(* IEC 61131-3 sources: teller/JD_Teller_LC2_V11/Class/Encoder_Inmeten, 1 file *)

(* ---- Encoder_Inmeten.st ---- *)
(*!
<Class
	Name               = "Encoder_Inmeten"
	Revision           = "0.0"
	RealtimeTask       = "false"
	CyclicTask         = "false"
	BackgroundTask     = "false"
	Sigmatek           = "false"
	OSInterface        = "false"
	HighPriority       = "false"
	Automatic          = "false"
	UpdateMode         = "Prescan"
	SharedCommandTable = "true"
	Objectsize         = "(570,120)">
	<Channels>
		<Server Name="ClassSvr" Visualized="false" Initialize="false" WriteProtected="true" Retentive="false"/>
		<Server Name="EncDiv" Visualized="true" Initialize="false" WriteProtected="true" Retentive="false"/>
		<Server Name="EncMul" Visualized="true" Initialize="false" WriteProtected="true" Retentive="false"/>
		<Server Name="ErrorEncDeltaIsNul" Visualized="true" Initialize="false" WriteProtected="true" Retentive="false"/>
		<Server Name="Lengte_MM" Visualized="true" Initialize="false" WriteProtected="false" Retentive="false"/>
		<Server Name="Reset" Visualized="true" Initialize="false" WriteProtected="false" Retentive="false"/>
		<Server Name="StartMeting" Visualized="true" Initialize="false" WriteProtected="false" Retentive="false"/>
		<Client Name="cEncoder" Required="true" Internal="false"/>
	</Channels>
</Class>
*)
Encoder_Inmeten : CLASS
  //Servers:
	ClassSvr 	: SvrChCmd_DINT;
	StartMeting 	: SvrCh_DINT;
	Lengte_MM 	: SvrCh_DINT;
	EncMul 	: SvrCh_DINT;
	EncDiv 	: SvrCh_DINT;
	Reset 	: SvrCh_DINT;
	ErrorEncDeltaIsNul 	: SvrCh_DINT;
  //Clients:
	cEncoder 	: CltCh_DINT;
  //Variables:
		EncoderStart 	: DINT;
  //Functions:

	FUNCTION VIRTUAL GLOBAL StartMeting::Write
		VAR_INPUT
			input (EAX) 	: DINT;
		END_VAR
		VAR_OUTPUT
			result (EAX) 	: DINT;
		END_VAR;

	FUNCTION VIRTUAL GLOBAL Lengte_MM::Write
		VAR_INPUT
			input (EAX) 	: DINT;
		END_VAR
		VAR_OUTPUT
			result (EAX) 	: DINT;
		END_VAR;

	FUNCTION VIRTUAL GLOBAL Reset::Write
		VAR_INPUT
			input (EAX) 	: DINT;
		END_VAR
		VAR_OUTPUT
			result (EAX) 	: DINT;
		END_VAR;
  //Tables:
	FUNCTION @STD
		VAR_OUTPUT
			ret_code	: CONFSTATES;
		END_VAR;
	FUNCTION GLOBAL TAB @CT_;
END_CLASS;

FUNCTION VIRTUAL GLOBAL Encoder_Inmeten::StartMeting::Write
	VAR_INPUT
		input (EAX) 	: DINT;
	END_VAR
	VAR_OUTPUT
		result (EAX) 	: DINT;
	END_VAR

	StartMeting := input;
  StartMeting := 1;

  cEncoder := cEncoder.Read();
  EncoderStart := cEncoder;

  //Init waardes Mul/Div
  EncDiv := 1000;
  EncMul := 0;
  Lengte_MM := 0;

	result := StartMeting;

END_FUNCTION

FUNCTION VIRTUAL GLOBAL Encoder_Inmeten::Lengte_MM::Write
	VAR_INPUT
		input (EAX) 	: DINT;
	END_VAR
	VAR_OUTPUT
		result (EAX) 	: DINT;
	END_VAR

  if    input < 1 then
        Lengte_MM := 1;
  else
        Lengte_MM := input;
  end_if;

  cEncoder := cEncoder.Read();

  if    cEncoder - EncoderStart = 0 then
        ErrorEncDeltaIsNul := 1;
        EncMul := 0;
  else
        ErrorEncDeltaIsNul := 0;
        EncMul := ((Lengte_MM * EncDiv) / abs(cEncoder - EncoderStart));
  end_if;

	result := Lengte_MM;

END_FUNCTION

FUNCTION VIRTUAL GLOBAL Encoder_Inmeten::Reset::Write
	VAR_INPUT
		input (EAX) 	: DINT;
	END_VAR
	VAR_OUTPUT
		result (EAX) 	: DINT;
	END_VAR

	Reset := input;

  StartMeting := 0;
  ErrorEncDeltaIsNul := 0;
  Lengte_MM := 0;
  EncDiv := 1000;
  EncMul := 0;

	result := Reset;

END_FUNCTION
